SUBAPPLICATION Uebung_010e_PC_B_OPC (* Geraet B (Station 12, 192.168.1.12): empfaengt Set/Reset/Toggle je per eigenem SERVER_0-Methodenaufruf (reiner RPC-Trigger, kein Wertwechsel-Trick, keine Bridge noetig), taktet die echte SR/Toggle-Flipflop-Logik (AX_T_FF_SR), schaltet DigitalOutput_Q1 und schreibt den neuen Zustand aktiv per CLIENT_1_0 zurueck auf Geraet A - 'SUB style': das Protokoll steckt im MyLib::sys-Composite, nicht in der Resource des Geraets *)
  (* Standard: 61499-2; Description: Copyright (c) 2026 Meisterschulen am Ostbahnhof This program and the accompanying materials are made available under the terms of the Eclipse Public License 2.0 which is available at https://www.eclipse.org/legal/epl-2.0/ SPDX-License-Identifier: EPL-2.0 *)
  (* Version 1.0, 2026-09-02, Franz Höpfinger, Meisterschulen am Ostbahnhof, initial API and implementation and/or initial documentation *)
  PACKAGE MyLib::sys;
  IMPORT logiBUS::io::DQ::logiBUS_DO;
  IMPORT logiBUS::io::DQ::logiBUS_DO_S;
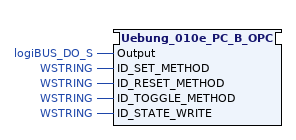
  VAR_INPUT
    Output : logiBUS::io::DQ::logiBUS_DO_S := logiBUS_DO::Invalid; (* Identify the Output Output_Q1..Q8 *)
    ID_SET_METHOD : WSTRING; (* Lokale Methodenadresse (ACTION=CREATE_METHOD) fuer den Set-Methodenaufruf, wird von Geraet A per CALL_METHOD aufgerufen *)
    ID_RESET_METHOD : WSTRING; (* Lokale Methodenadresse (ACTION=CREATE_METHOD) fuer den Reset-Methodenaufruf, wird von Geraet A per CALL_METHOD aufgerufen *)
    ID_TOGGLE_METHOD : WSTRING; (* Lokale Methodenadresse (ACTION=CREATE_METHOD) fuer den Toggle-Methodenaufruf, wird von Geraet A per CALL_METHOD aufgerufen *)
    ID_STATE_WRITE : WSTRING; (* Remote-Ziel-Adresse (BOOL, ACTION=WRITE) fuer den Flipflop-Zustand auf Geraet A *)
  END_VAR
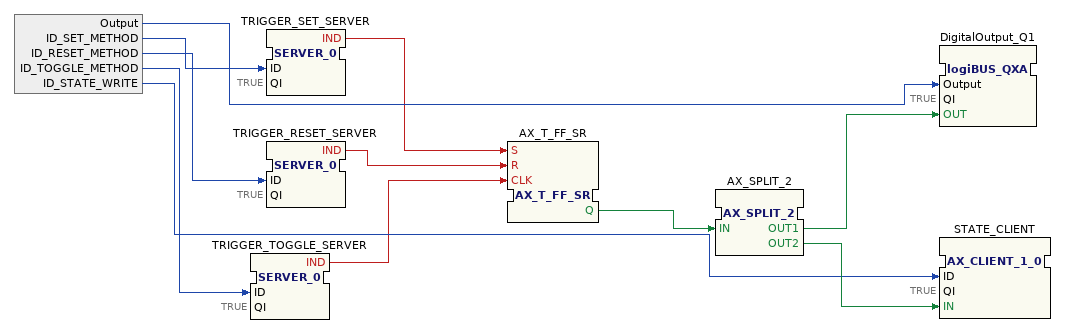
  FBS
    TRIGGER_SET_SERVER : iec61499::net::SERVER_0(QI := TRUE);
    TRIGGER_RESET_SERVER : iec61499::net::SERVER_0(QI := TRUE);
    TRIGGER_TOGGLE_SERVER : iec61499::net::SERVER_0(QI := TRUE);
    AX_T_FF_SR : adapter::events::unidirectional::AX_T_FF_SR;
    AX_SPLIT_2 : adapter::events::unidirectional::AX_SPLIT_2;
    DigitalOutput_Q1 : logiBUS::io::DQ::logiBUS_QXA(QI := TRUE);
    STATE_CLIENT : adapter::net::AX_CLIENT_1_0(QI := TRUE);
  END_FBS
  EVENT_CONNECTIONS
    TRIGGER_SET_SERVER.IND TO AX_T_FF_SR.S;
    TRIGGER_RESET_SERVER.IND TO AX_T_FF_SR.R;
    TRIGGER_TOGGLE_SERVER.IND TO AX_T_FF_SR.CLK;
  END_CONNECTIONS
  DATA_CONNECTIONS
    Output TO DigitalOutput_Q1.Output;
    ID_SET_METHOD TO TRIGGER_SET_SERVER.ID;
    ID_RESET_METHOD TO TRIGGER_RESET_SERVER.ID;
    ID_TOGGLE_METHOD TO TRIGGER_TOGGLE_SERVER.ID;
    ID_STATE_WRITE TO STATE_CLIENT.ID;
  END_CONNECTIONS
  ADAPTER_CONNECTIONS
    AX_T_FF_SR.Q TO AX_SPLIT_2.IN;
    AX_SPLIT_2.OUT1 TO DigitalOutput_Q1.OUT;
    AX_SPLIT_2.OUT2 TO STATE_CLIENT.IN;
  END_CONNECTIONS
END_SUBAPPLICATION
